Universal Robots PolyScope program: calibration.urp

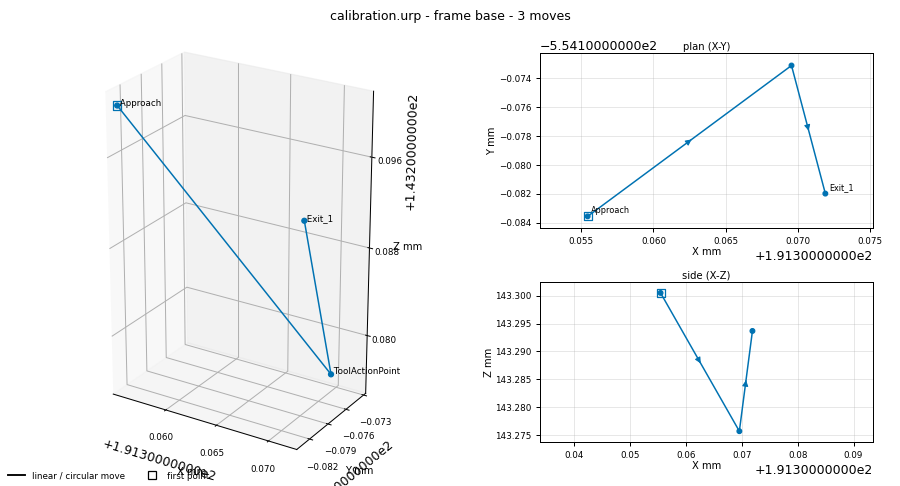
[picture p0: tool path of calibration.urp in frame base, 3 of 3 moves have a stored position in this frame; points joined in program order, loops and branches not executed]
Program calibration (installation=default directory=/programs/HandEyeCalibration createdIn=3.10.1.76190 lastSavedIn=5.9.1.1031110 robotSerialNumber=20185500256)
Calibrated DH parameters: a=[0.000163, -0.146131, -0.38577, 0.000126, -0.000021, 0]; d=[0.161954, 188.306531, -157.478086, -30.695088, 0.099716, 0.099628]; alpha=[1.569701, -0.00212, 0.002263, 1.570438, -1.570123, 0]; deltaTheta=[0, -1.219859, 7.681919, -0.178877, -0.000001, 0]
BeforeStart
  SuppressedNode
    recorder := rpc_factory("xmlrpc", "http://192.168.1.119:10000")
Robot Program (runOnlyOnce=true)
  Loop Counting (count=24) loopVariable(name=Loop_1)
    URCap Palletizing (pallet-impl, Universal Robots) dataModel(palletFeature=Base, isPalletizing=true, Length(key=objectHeight value=0.05 unit=M), Variable(key=name, variable(name=Pallet_1)), Variable(key=globalCountingVariable, variable(name=Pallet_1_cnt, initializeExpression=1)), Variable(key=layerNumberVariable, variable(name=Pallet_1_lno, initializeExpression=1)), Variable(key=layerCountingVariable, variable(name=Pallet_1_lct, initializeExpression=1)), Variable(key=handleSeparatorVariable, variable(name=Pallet_1_sep, initializeExpression=False)), Variable(key=totalCountVariable, variable(name=Pallet_1_tct, initializeExpression=1)), Variable(key=referencePoint, variable(featureName=referencePoint)), Variable(key=separatorPoint, variable(featureName=separatorPoint))); state(isChildrenLocked=true)
      URCap Patterns (pallet-impl, Universal Robots) state(isChildrenLocked=true)
        URCap Pattern (pallet-impl, Universal Robots) dataModel(UUID=3b75a608-283e-4ba5-887e-097f98334a24, patternType=GRID, rows=6, columns=4, Variable(key=nameVariable, variable(name=Grid_Pattern_1))); state(isChildrenLocked=true)
          URCap Item (pallet-impl, Universal Robots) dataModel(UUID=c9c99c67-97d1-430b-a99c-1a147d52fbce, patternType=GRID, index=0, calibrationDeltaTheta=[5.766864417944273E-8, -1.219858784201824, 7.681919015479748, -0.17887715072020058, -5.825955228730417E-7, 1.2463722892999685E-7], calibrationA=[1.6278795868896034E-4, -0.14613148603940784, -0.3857702315473692, 1.264637573695105E-4, -2.1298401427010558E-5, 0.0], calibrationD=[0.16195415116355033, 188.3065313778212, -157.47808565825918, -30.695087710514088, 0.09971634582834017, 0.09962824424434498], calibrationAlpha=[1.5697008015899263, -0.0021197873275575997, 0.0022625217605951827, 1.5704375006736107, -1.570122774022032, 0.0], calibrationJointChecksum=[-1856353559, -1856958578, 625087103, -1528685046, -1528462798, -1527923809], calibrationStatus=2, calibrationValidChecksum=true, baseToFeature=[0.0, 0.0, 0.0, 0.0, 0.0, 0.0], TCPOffset=[-1.0286583455310083E-5, -1.815219158174397E-5, 0.2504943115515415, 2.3863615101507944E-6, 1.2142012508486024E-5, 2.1928973603070405E-5], Variable(key=variable, variable(name=CornerItem_1)), JointPositions(key=jointpositions, JointPosition(key=[1], Angle(key=pos value=1.829047 unit=RAD)), JointPosition(key=[2], Angle(key=pos value=-1.014036 unit=RAD)), JointPosition(key=[3], Angle(key=pos value=1.084977 unit=RAD)), JointPosition(key=[4], Angle(key=pos value=-1.267398 unit=RAD)), JointPosition(key=[5], Angle(key=pos value=-1.830007 unit=RAD)), JointPosition(key=[6], Angle(key=pos value=2.369849 unit=RAD))))
          URCap Item (pallet-impl, Universal Robots) dataModel(UUID=f56a354f-8c68-413d-8676-7945f6eb2195, patternType=GRID, index=1, calibrationDeltaTheta=[5.766864417944273E-8, -1.219858784201824, 7.681919015479748, -0.17887715072020058, -5.825955228730417E-7, 1.2463722892999685E-7], calibrationA=[1.6278795868896034E-4, -0.14613148603940784, -0.3857702315473692, 1.264637573695105E-4, -2.1298401427010558E-5, 0.0], calibrationD=[0.16195415116355033, 188.3065313778212, -157.47808565825918, -30.695087710514088, 0.09971634582834017, 0.09962824424434498], calibrationAlpha=[1.5697008015899263, -0.0021197873275575997, 0.0022625217605951827, 1.5704375006736107, -1.570122774022032, 0.0], calibrationJointChecksum=[-1856353559, -1856958578, 625087103, -1528685046, -1528462798, -1527923809], calibrationStatus=2, calibrationValidChecksum=true, baseToFeature=[0.0, 0.0, 0.0, 0.0, 0.0, 0.0], TCPOffset=[1.853792899625395E-5, 1.1078837976574718E-5, 0.2505141323808394, -9.051397742641462E-6, -1.6129430841377793E-5, -2.3493589080937635E-5], Variable(key=variable, variable(name=CornerItem_2)), JointPositions(key=jointpositions, JointPosition(key=[1], Angle(key=pos value=0.98484 unit=RAD)), JointPosition(key=[2], Angle(key=pos value=-0.994288 unit=RAD)), JointPosition(key=[3], Angle(key=pos value=0.980622 unit=RAD)), JointPosition(key=[4], Angle(key=pos value=-1.129374 unit=RAD)), JointPosition(key=[5], Angle(key=pos value=-1.41382 unit=RAD)), JointPosition(key=[6], Angle(key=pos value=3.278991 unit=RAD))))
          URCap Item (pallet-impl, Universal Robots) dataModel(UUID=3829da42-c55d-4a5c-b457-f64e555102c7, patternType=GRID, index=2, calibrationDeltaTheta=[5.766864417944273E-8, -1.219858784201824, 7.681919015479748, -0.17887715072020058, -5.825955228730417E-7, 1.2463722892999685E-7], calibrationA=[1.6278795868896034E-4, -0.14613148603940784, -0.3857702315473692, 1.264637573695105E-4, -2.1298401427010558E-5, 0.0], calibrationD=[0.16195415116355033, 188.3065313778212, -157.47808565825918, -30.695087710514088, 0.09971634582834017, 0.09962824424434498], calibrationAlpha=[1.5697008015899263, -0.0021197873275575997, 0.0022625217605951827, 1.5704375006736107, -1.570122774022032, 0.0], calibrationJointChecksum=[-1856353559, -1856958578, 625087103, -1528685046, -1528462798, -1527923809], calibrationStatus=2, calibrationValidChecksum=true, baseToFeature=[0.0, 0.0, 0.0, 0.0, 0.0, 0.0], TCPOffset=[-2.638578009794834E-5, -1.1109026301692193E-5, 0.25052083345408926, 1.2465270259924581E-5, -6.508066330076159E-5, -2.4633615436690955E-5], Variable(key=variable, variable(name=CornerItem_3)), JointPositions(key=jointpositions, JointPosition(key=[1], Angle(key=pos value=0.382995 unit=RAD)), JointPosition(key=[2], Angle(key=pos value=-1.838224 unit=RAD)), JointPosition(key=[3], Angle(key=pos value=2.000757 unit=RAD)), JointPosition(key=[4], Angle(key=pos value=-1.442862 unit=RAD)), JointPosition(key=[5], Angle(key=pos value=-1.194043 unit=RAD)), JointPosition(key=[6], Angle(key=pos value=4.066689 unit=RAD))))
          URCap Item (pallet-impl, Universal Robots) dataModel(UUID=a3c91444-18ff-48ff-82e8-cf9579b0eb98, patternType=GRID, index=3, calibrationDeltaTheta=[5.766864417944273E-8, -1.219858784201824, 7.681919015479748, -0.17887715072020058, -5.825955228730417E-7, 1.2463722892999685E-7], calibrationA=[1.6278795868896034E-4, -0.14613148603940784, -0.3857702315473692, 1.264637573695105E-4, -2.1298401427010558E-5, 0.0], calibrationD=[0.16195415116355033, 188.3065313778212, -157.47808565825918, -30.695087710514088, 0.09971634582834017, 0.09962824424434498], calibrationAlpha=[1.5697008015899263, -0.0021197873275575997, 0.0022625217605951827, 1.5704375006736107, -1.570122774022032, 0.0], calibrationJointChecksum=[-1856353559, -1856958578, 625087103, -1528685046, -1528462798, -1527923809], calibrationStatus=2, calibrationValidChecksum=true, baseToFeature=[0.0, 0.0, 0.0, 0.0, 0.0, 0.0], TCPOffset=[-1.6622661828114005E-5, -9.212937447378167E-7, 0.25049158554484907, -1.3763171141184998E-5, -1.8353878957609274E-5, -1.3926437959700817E-5], Variable(key=variable, variable(name=CornerItem_4)), JointPositions(key=jointpositions, JointPosition(key=[1], Angle(key=pos value=2.115002 unit=RAD)), JointPosition(key=[2], Angle(key=pos value=-1.842088 unit=RAD)), JointPosition(key=[3], Angle(key=pos value=2.096842 unit=RAD)), JointPosition(key=[4], Angle(key=pos value=-1.912626 unit=RAD)), JointPosition(key=[5], Angle(key=pos value=-2.019257 unit=RAD)), JointPosition(key=[6], Angle(key=pos value=1.445286 unit=RAD))))
      URCap Layers (pallet-impl, Universal Robots) dataModel(separators=[false], selectedPatterns=[3b75a608-283e-4ba5-887e-097f98334a24])
      URCap At Each Item (pallet-impl, Universal Robots) dataModel(selectedPattern=3b75a608-283e-4ba5-887e-097f98334a24, selectedPosition=c9c99c67-97d1-430b-a99c-1a147d52fbce, Approach_calibrationDeltaTheta=[5.766864417944273E-8, -1.219858784201824, 7.681919015479748, -0.17887715072020058, -5.825955228730417E-7, 1.2463722892999685E-7], Approach_calibrationA=[1.6278795868896034E-4, -0.14613148603940784, -0.3857702315473692, 1.264637573695105E-4, -2.1298401427010558E-5, 0.0], Approach_calibrationD=[0.16195415116355033, 188.3065313778212, -157.47808565825918, -30.695087710514088, 0.09971634582834017, 0.09962824424434498], Approach_calibrationAlpha=[1.5697008015899263, -0.0021197873275575997, 0.0022625217605951827, 1.5704375006736107, -1.570122774022032, 0.0], Approach_calibrationJointChecksum=[-1856353559, -1856958578, 625087103, -1528685046, -1528462798, -1527923809], Approach_calibrationStatus=2, Approach_calibrationValidChecksum=true, Approach_baseToFeature=[0.0, 0.0, 0.0, 0.0, 0.0, 0.0], Approach_TCPOffset=[-1.3892902311629651E-5, -1.773570889707088E-5, 0.2504796854129975, 4.54528904575002E-7, -6.683241556042285E-5, -1.1448191040776278E-5], Exit_calibrationDeltaTheta=[5.766864417944273E-8, -1.219858784201824, 7.681919015479748, -0.17887715072020058, -5.825955228730417E-7, 1.2463722892999685E-7], Exit_calibrationA=[1.6278795868896034E-4, -0.14613148603940784, -0.3857702315473692, 1.264637573695105E-4, -2.1298401427010558E-5, 0.0], Exit_calibrationD=[0.16195415116355033, 188.3065313778212, -157.47808565825918, -30.695087710514088, 0.09971634582834017, 0.09962824424434498], Exit_calibrationAlpha=[1.5697008015899263, -0.0021197873275575997, 0.0022625217605951827, 1.5704375006736107, -1.570122774022032, 0.0], Exit_calibrationJointChecksum=[-1856353559, -1856958578, 625087103, -1528685046, -1528462798, -1527923809], Exit_calibrationStatus=2, Exit_calibrationValidChecksum=true, Exit_baseToFeature=[0.0, 0.0, 0.0, 0.0, 0.0, 0.0], Exit_TCPOffset=[-5.1097214677775504E-6, -2.205200201554902E-6, 0.25048063657230407, -3.306392049443238E-5, -3.223041893091702E-5, 2.4770728605915508E-5], currentWizardState=LANDING, Pose(key=refBaseToFeature, Position(key=posePosition, Length(key=X value=0 unit=M), Length(key=Y value=0 unit=M), Length(key=Z value=0 unit=M)), Rotation(key=poseRotation, Angle(key=RX value=0 unit=RAD), Angle(key=RY value=0 unit=RAD), Angle(key=RZ value=0 unit=RAD))), Pose(key=refPose, Position(key=posePosition, Length(key=X value=0.19137 unit=M), Length(key=Y value=-0.554173 unit=M), Length(key=Z value=0.143276 unit=M)), Rotation(key=poseRotation, Angle(key=RX value=-2.322171 unit=RAD), Angle(key=RY value=-1.394433 unit=RAD), Angle(key=RZ value=0.215065 unit=RAD))), JointPositions(key=Approach_jointpositions, JointPosition(key=[1], Angle(key=pos value=1.829019 unit=RAD)), JointPosition(key=[2], Angle(key=pos value=-1.014043 unit=RAD)), JointPosition(key=[3], Angle(key=pos value=1.084958 unit=RAD)), JointPosition(key=[4], Angle(key=pos value=-1.267368 unit=RAD)), JointPosition(key=[5], Angle(key=pos value=-1.83001 unit=RAD)), JointPosition(key=[6], Angle(key=pos value=2.369846 unit=RAD))), JointPositions(key=Exit_jointpositions, JointPosition(key=[1], Angle(key=pos value=1.829019 unit=RAD)), JointPosition(key=[2], Angle(key=pos value=-1.014043 unit=RAD)), JointPosition(key=[3], Angle(key=pos value=1.084958 unit=RAD)), JointPosition(key=[4], Angle(key=pos value=-1.267368 unit=RAD)), JointPosition(key=[5], Angle(key=pos value=-1.83001 unit=RAD)), JointPosition(key=[6], Angle(key=pos value=2.369846 unit=RAD))))
        URCap Generated Movements (pallet-impl, Universal Robots) state(isChildrenLocked=true)
          MoveJ speed 60 deg/s, acceleration 80 deg/s^2 (useActiveTCP=true) feature=referencePoint
            Waypoint Approach: TCP in base x=191.355 y=-554.184 z=143.3 mm, rx=-2.3222 ry=-1.3945 rz=0.2151 rad; joints [98.75, -58.705, 99.882, -111.335, -107, 129.981] deg; TCP offset x=0 y=0 z=0 mm, rx=0 ry=0 rz=0 rad; feature pose in base x=191.37 y=-554.173 z=143.276 mm, rx=-2.3222 ry=-1.3944 rz=0.2151 rad
          MoveL speed 250 mm/s, acceleration 1200 mm/s^2 (useActiveTCP=true) feature(featureName=referencePoint)
            Waypoint ToolActionPoint: TCP in base x=191.37 y=-554.173 z=143.276 mm, rx=-2.3222 ry=-1.3944 rz=0.2151 rad; joints [98.751, -58.704, 99.882, -111.334, -106.997, 129.983] deg; TCP offset x=0 y=0 z=0 mm, rx=0 ry=0 rz=0 rad
          Folder Tool action
            Wait Sleep waitTime=1
          MoveL speed 250 mm/s, acceleration 1200 mm/s^2 (useActiveTCP=true) feature(featureName=referencePoint)
            Waypoint Exit_1: TCP in base x=191.372 y=-554.182 z=143.294 mm, rx=-2.3222 ry=-1.3944 rz=0.2151 rad; joints [98.751, -58.705, 99.881, -111.335, -106.997, 129.984] deg; TCP offset x=0 y=0 z=0 mm, rx=0 ry=0 rz=0 rad
SuppressedNode
  SubProgram send_pose (keepSynchronizedWithDisk=false)
    Wait Sleep waitTime=0.5
    Wait Condition expression=is_steady()
    handle := recorder.add_sample(get_actual_tool_flange_pose())
